PROGRAM MB_CLIENT_DEMO
VAR
	IP_CONTROL2_1: IP_CONTROL2;
	MB_CLIENT_1: MB_CLIENT;
	IP_C: IP_C;
	S_BUF: NETWORK_BUFFER_SHORT;
	R_BUF: NETWORK_BUFFER_SHORT;
	DATA: ARRAY [0..255] OF WORD;
	W_DATA_BITPOS: INT;
	W_DATA_ADR: INT;
	W_POINTS: INT;
	W_ADDR: INT;
	R_DATA_BITPOS: INT;
	R_DATA_ADR: INT;
	R_POINTS: INT;
	R_ADDR: INT;
	FC: INT;
	ENABLE: BOOL;
END_VAR
VAR // added by the converter: edge detectors and wires of the graphical bodies
    _w1 : ANY;
END_VAR

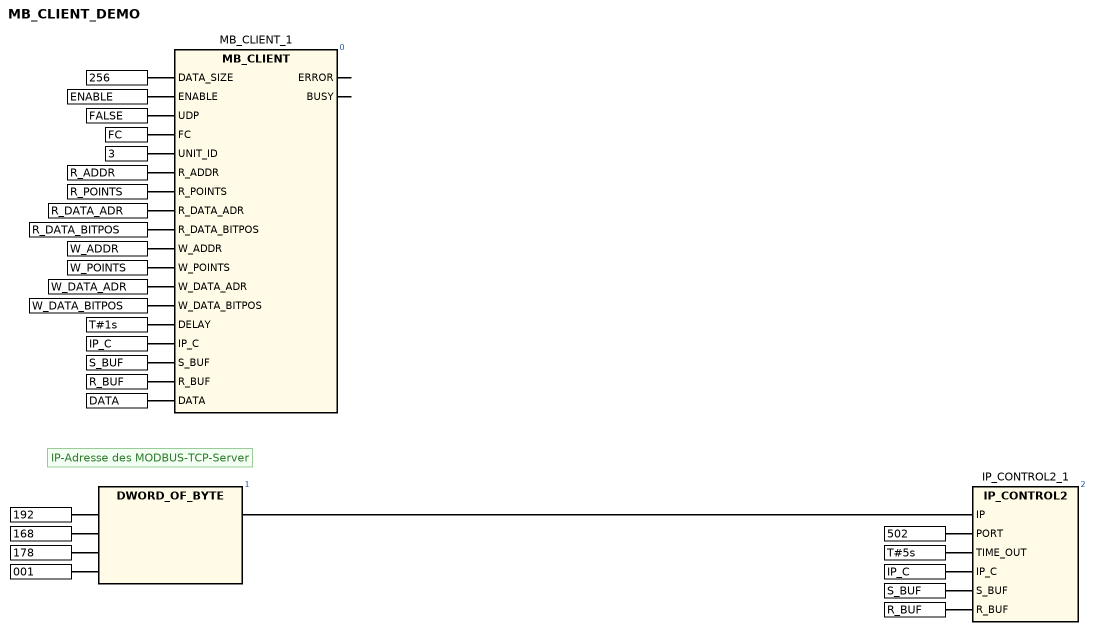
MB_CLIENT_1(
    DATA_SIZE := 256,
    ENABLE := ENABLE,
    UDP := FALSE,
    FC := FC,
    UNIT_ID := 3,
    R_ADDR := R_ADDR,
    R_POINTS := R_POINTS,
    R_DATA_ADR := R_DATA_ADR,
    R_DATA_BITPOS := R_DATA_BITPOS,
    W_ADDR := W_ADDR,
    W_POINTS := W_POINTS,
    W_DATA_ADR := W_DATA_ADR,
    W_DATA_BITPOS := W_DATA_BITPOS,
    DELAY := T#1s,
    IP_C := IP_C,
    S_BUF := S_BUF,
    R_BUF := R_BUF,
    DATA := DATA); // MB_CLIENT
// IP-Adresse des MODBUS-TCP-Server
_w1 := DWORD_OF_BYTE(192, 168, 178, 001);
IP_CONTROL2_1(IP := _w1, PORT := 502, TIME_OUT := T#5s, IP_C := IP_C, S_BUF := S_BUF, R_BUF := R_BUF); // IP_CONTROL2

END_PROGRAM

(* stored: Version 1.1.0.1, ProductVersion 3.1.4022.7
   POU MB_CLIENT_DEMO: Id {30e86327-f0dd-422c-ab01-e649441fd88e}, SpecialFunc None *)
